// TIA Portal V20 export
DATA_BLOCK "DB_BwLoader"   // DB108
// stored: InstanceOfName FB_BwLoader, InstanceOfType FB
"FB_BwLoader"
   // VAR
   //    sBwCommunication : "FB_BwCommunication";
   //    sTONBW_CtrlInProgress { S7_SetPoint := 'True'} : TP_TIME;
   // END_VAR
BEGIN
END_DATA_BLOCK
